// TIA Portal V20 export
FUNCTION_BLOCK "05 T1-A ARUNC Sequence"   // FB1502, GRAPH
// stored: AutoNumber false, GraphVersion 6.0, InitialValuesAcquisition false, SetENOAutomatically false
   // inherited from GRAPH_BASE
   VAR_INPUT
      OFF_SQ : Bool := false;
      INIT_SQ : Bool := false;
      ACK_EF : Bool := false;
      S_PREV : Bool := false;
      S_NEXT : Bool := false;
      SW_AUTO : Bool := false;
      SW_TAP : Bool := false;
      SW_TOP : Bool := false;
      SW_MAN : Bool := false;
      S_SEL : Int := 0;
      S_ON : Bool := false;
      S_OFF : Bool := false;
      T_PUSH : Bool := false;
   END_VAR
   VAR_OUTPUT
      S_NO : Int := 0;
      S_MORE : Bool := false;
      S_ACTIVE : Bool := false;
      ERR_FLT : Bool := false;
      AUTO_ON : Bool := false;
      TAP_ON : Bool := false;
      TOP_ON : Bool := false;
      MAN_ON : Bool := false;
   END_VAR
BEGIN
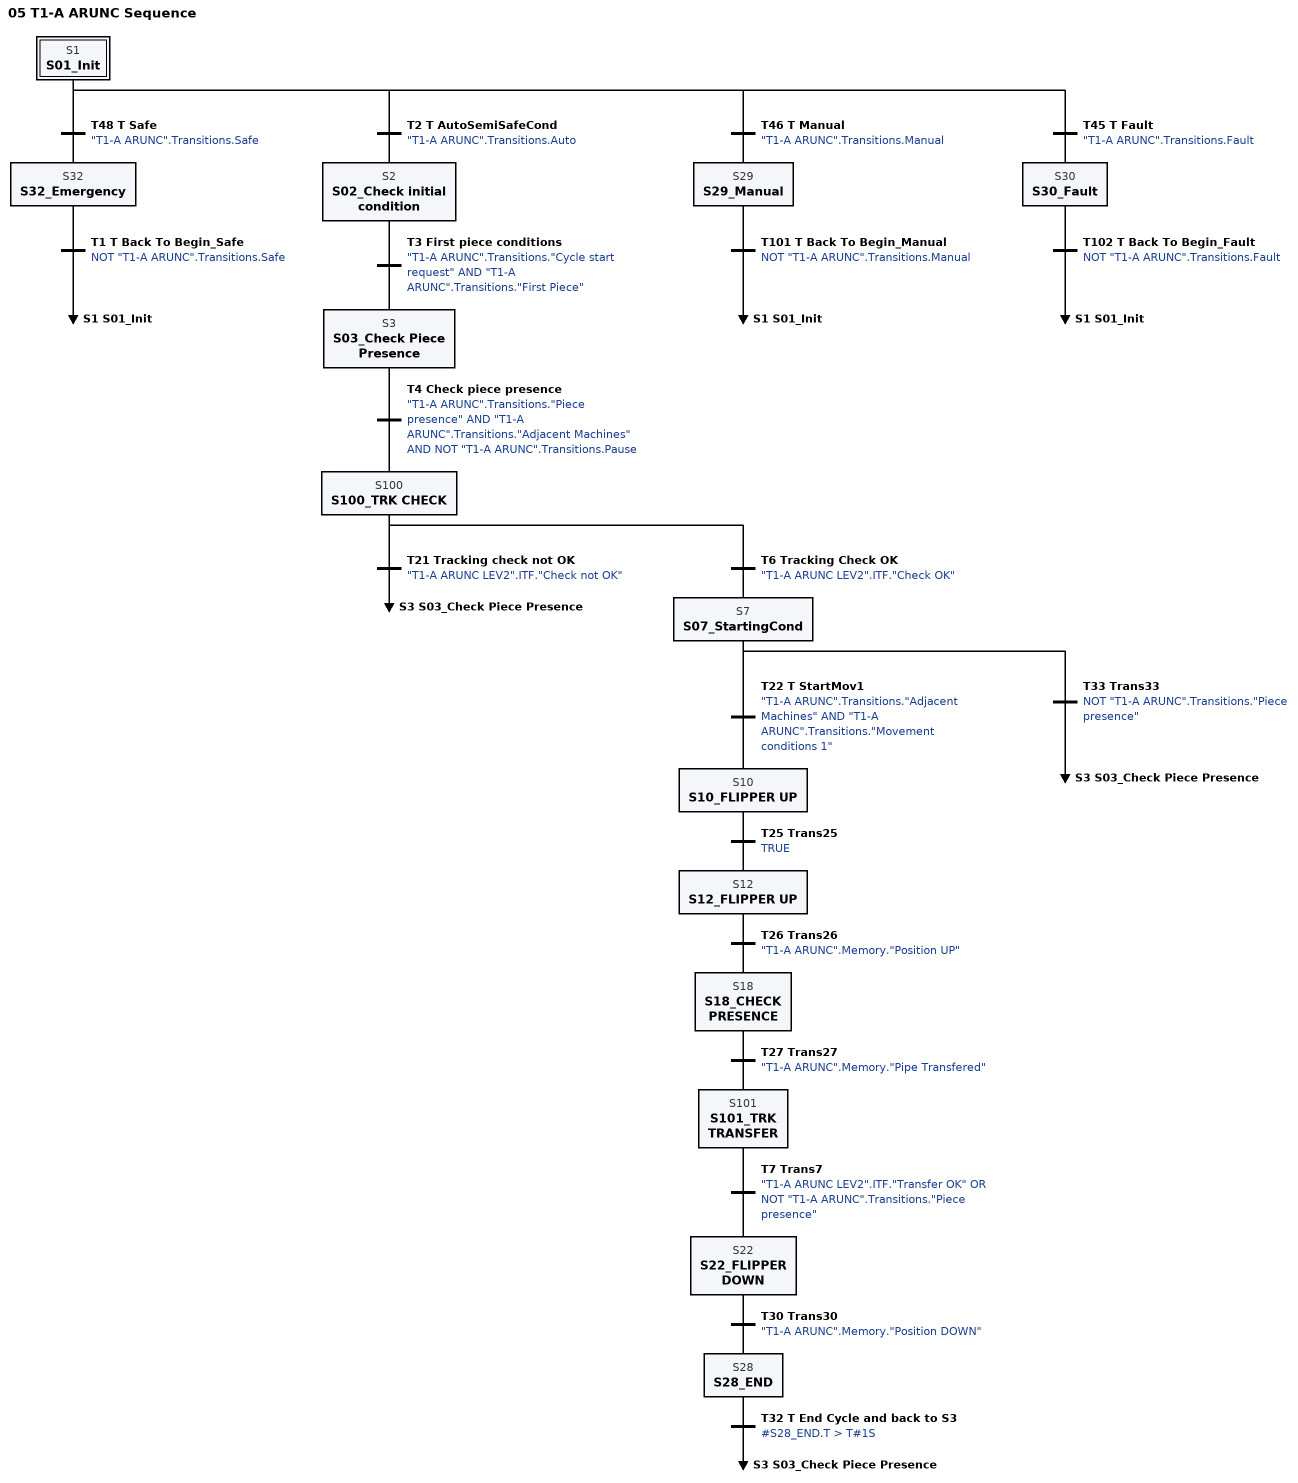
   // permanent pre-instructions
   NETWORK 1
      "01 T1-A ARUNC Alarms"();
   NETWORK 2
      "02 T1-A ARUNC HMI"();
   NETWORK 3
      "03 T1-A ARUNC Aux"();
   NETWORK 4
      "04 T1-A ARUNC Transitions"();

   // sequencer 1
   INITIAL_STEP S01_Init:   // S1, max time T#10S, warning time T#7S
   END_STEP
   TRANSITION "T Safe" FROM S01_Init TO S32_Emergency   // T48
      := "T1-A ARUNC".Transitions.Safe;
   END_TRANSITION
   TRANSITION "T AutoSemiSafeCond" FROM S01_Init TO "S02_Check initial condition"   // T2
      := "T1-A ARUNC".Transitions.Auto;
   END_TRANSITION
   TRANSITION "T Manual" FROM S01_Init TO S29_Manual   // T46
      := "T1-A ARUNC".Transitions.Manual;
   END_TRANSITION
   TRANSITION "T Fault" FROM S01_Init TO S30_Fault   // T45
      := "T1-A ARUNC".Transitions.Fault;
   END_TRANSITION
   STEP "S03_Check Piece Presence":   // S3, max time T#10S, warning time T#7S
   END_STEP
   TRANSITION "Check piece presence" FROM "S03_Check Piece Presence" TO "S100_TRK CHECK"   // T4
      := "T1-A ARUNC".Transitions."Piece presence" AND "T1-A ARUNC".Transitions."Adjacent Machines" AND NOT "T1-A ARUNC".Transitions.Pause;
   END_TRANSITION
   STEP S32_Emergency:   // S32, max time T#10S, warning time T#7S
   END_STEP
   TRANSITION "T Back To Begin_Safe" FROM S32_Emergency TO S01_Init   // T1, jump
      := NOT "T1-A ARUNC".Transitions.Safe;
   END_TRANSITION
   STEP S29_Manual:   // S29, max time T#10S, warning time T#7S
   END_STEP
   TRANSITION "T Back To Begin_Manual" FROM S29_Manual TO S01_Init   // T101, jump
      := NOT "T1-A ARUNC".Transitions.Manual;
   END_TRANSITION
   STEP "S02_Check initial condition":   // S2, max time T#10S, warning time T#7S
   END_STEP
   TRANSITION "First piece conditions" FROM "S02_Check initial condition" TO "S03_Check Piece Presence"   // T3
      := "T1-A ARUNC".Transitions."Cycle start request" AND "T1-A ARUNC".Transitions."First Piece";
   END_TRANSITION
   STEP S30_Fault:   // S30, max time T#10S, warning time T#7S
   END_STEP
   TRANSITION "T Back To Begin_Fault" FROM S30_Fault TO S01_Init   // T102, jump
      := NOT "T1-A ARUNC".Transitions.Fault;
   END_TRANSITION
   STEP S28_END:   // S28, max time T#10S, warning time T#7S
   END_STEP
   TRANSITION "T End Cycle and back to S3" FROM S28_END TO "S03_Check Piece Presence"   // T32, jump: Assenza pezzo o ok da robot
      := #S28_END.T > T#1S;
   END_TRANSITION
   STEP "S10_FLIPPER UP":   // S10, max time T#10S, warning time T#7S
   END_STEP
   TRANSITION Trans25 FROM "S10_FLIPPER UP" TO "S12_FLIPPER UP"   // T25
      := TRUE;
   END_TRANSITION
   STEP "S12_FLIPPER UP":   // S12, max time T#10S, warning time T#7S
   END_STEP
   TRANSITION Trans26 FROM "S12_FLIPPER UP" TO "S18_CHECK PRESENCE"   // T26
      := "T1-A ARUNC".Memory."Position UP";
   END_TRANSITION
   STEP "S18_CHECK PRESENCE":   // S18, max time T#10S, warning time T#7S
   END_STEP
   TRANSITION Trans27 FROM "S18_CHECK PRESENCE" TO "S101_TRK TRANSFER"   // T27
      := "T1-A ARUNC".Memory."Pipe Transfered";
   END_TRANSITION
   STEP "S100_TRK CHECK":   // S100, max time T#10S, warning time T#7S
   END_STEP
   TRANSITION "Tracking check not OK" FROM "S100_TRK CHECK" TO "S03_Check Piece Presence"   // T21, jump
      := "T1-A ARUNC LEV2".ITF."Check not OK";
   END_TRANSITION
   TRANSITION "Tracking Check OK" FROM "S100_TRK CHECK" TO S07_StartingCond   // T6
      := "T1-A ARUNC LEV2".ITF."Check OK";
   END_TRANSITION
   STEP "S22_FLIPPER DOWN":   // S22, max time T#10S, warning time T#7S
   END_STEP
   TRANSITION Trans30 FROM "S22_FLIPPER DOWN" TO S28_END   // T30
      := "T1-A ARUNC".Memory."Position DOWN";
   END_TRANSITION
   STEP "S101_TRK TRANSFER":   // S101, max time T#10S, warning time T#7S
   END_STEP
   TRANSITION Trans7 FROM "S101_TRK TRANSFER" TO "S22_FLIPPER DOWN"   // T7
      := "T1-A ARUNC LEV2".ITF."Transfer OK" OR NOT "T1-A ARUNC".Transitions."Piece presence";
   END_TRANSITION
   STEP S07_StartingCond:   // S7, max time T#10S, warning time T#7S
   END_STEP
   TRANSITION "T StartMov1" FROM S07_StartingCond TO "S10_FLIPPER UP"   // T22
      := "T1-A ARUNC".Transitions."Adjacent Machines" AND "T1-A ARUNC".Transitions."Movement conditions 1";
   END_TRANSITION
   TRANSITION Trans33 FROM S07_StartingCond TO "S03_Check Piece Presence"   // T33, jump
      := NOT "T1-A ARUNC".Transitions."Piece presence";
   END_TRANSITION

   // permanent post-instructions
   NETWORK 1
      "06 T1-A ARUNC Output"();
   NETWORK 2
      "07 T1-A ARUNC LEV2"();
END_FUNCTION_BLOCK
